INTERFACE I_ActuatorLeftRight EXTENDS I_ActuatorBase

{attribute 'monitoring' := 'call'}
PROPERTY public leftOk : BOOL
GET
END_GET
END_PROPERTY

{attribute 'monitoring' := 'call'}
PROPERTY public rightOk : BOOL
GET
END_GET
END_PROPERTY

METHOD public toTheLeft : BOOL
VAR_INPUT
END_VAR
END_METHOD

METHOD public toTheRight : BOOL
VAR_INPUT
END_VAR
END_METHOD

END_INTERFACE

(* stored: Version 1.1.0.1, ProductVersion 3.1.4024.3
   Itf I_ActuatorLeftRight: Id {9368650c-3cf5-460f-88e3-a1983b984127}
   Property leftOk: Id {3f4df3b8-23c1-4781-b59a-8391e2d92380}
   Get Get: Id {ccc850b2-dc49-40c9-bd79-a90f670c7781}
   Property rightOk: Id {4519aa7e-24dc-45bd-9ad8-819f5b8862cb}
   Get Get: Id {ffe09f00-adda-4120-92b0-b58f41975e55}
   Method toTheLeft: Id {f101f148-5fe7-4664-a45f-10c8281df8fb}
   Method toTheRight: Id {a80bbd77-0f93-4064-a024-3a79428d4c7c} *)
